KUKA KRL program: dockof_1.src, dockof_1.dat

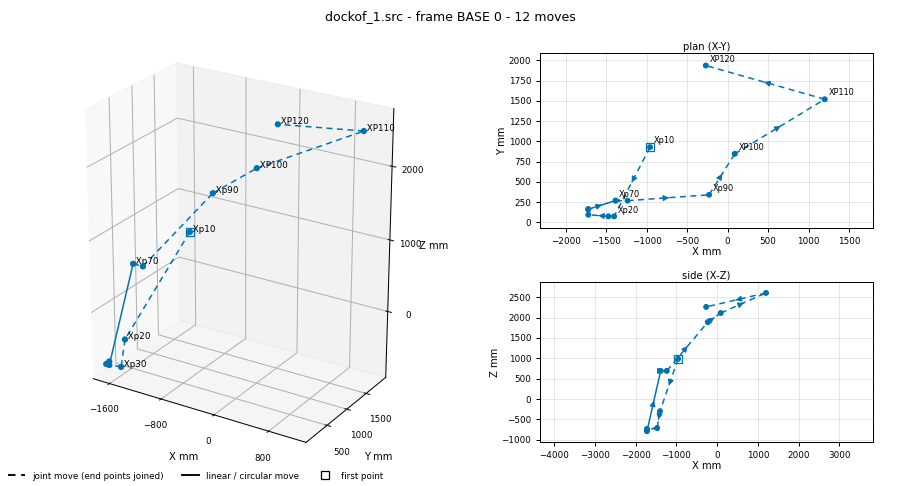
[picture p0: tool path of dockof_1.src in frame BASE 0, 12 of 12 moves have a stored position in this frame; points joined in program order, loops and branches not executed]
--- dockof_1.src ---
&ACCESS RVP1
&REL 140
&COMMENT PLACE GUN 1
DEF DOCKOF_1( )
;================================================
; MODEL    :
; IE GROUP :
; STATION  :
; ROBOT    :
; FUNCTION : DOCK OFF GUN 1
;================================================
;FOLD INI
;FOLD BASISTECH INI
GLOBAL INTERRUPT DECL 3 WHEN $STOPMESS==TRUE DO IR_STOPM ( )
INTERRUPT ON 3
BAS (#INITMOV,0 )
;ENDFOLD (BASISTECH INI)
;FOLD GRIPPERTECH INI
USER_GRP(0,DUMMY,DUMMY,GDEFAULT)
;ENDFOLD (GRIPPERTECH INI)
;FOLD USER INI
;Make your modifications here

;ENDFOLD (USER INI)
;ENDFOLD (INI)

PGNO1_TYPE=0

;FOLD PTP p10 H RETR CLS Gun= 1 Pair= FIRST Tool[1]:Gun 1 Base[0];%{PE}%R 6.0.16,%MKUKATPSPOT,%CRETR,%VPTP,%P 1:PTP, 2:p10, 3:, 5:100, 7:H, 9:#CLO, 11:1, 13:#FIRST
$BWDSTART=FALSE
PDAT_ACT=PH
FDAT_ACT=Fp10
BAS(#PTP_PARAMS,PH.VEL)
S_ACT.GUN=1
S_ACT.PAIR=#FIRST
S_ACT.RETR=#CLO
S_READY=FALSE
TRIGGER WHEN DISTANCE=1 DELAY=0.0 DO USERSPOT(#RETR, S_ACT) PRIO=-1
PTP Xp10
WAIT FOR S_READY
;ENDFOLD

;Open flap 1
;FOLD DOCKING.FLAP_OPN 1 ;%{PE}%MKUKATPUSER
DOCKING (#FLAP_OPN ,1)
;ENDFOLD

;FOLD ; Check docking station 1 ready to dock off;%{PE}%R 2.4.14,%MKUKATPBASIS,%CCOMMENT,%VNORMAL,%P 2:Check docking station 1 ready to dock off
;ENDFOLD
DOCKING (#REQ_DOCK_OFF,1)

;FOLD PTP p20 CONT Vel= 100 % H Tool[1]:Gun 1 Base[0];%{PE}%R 5.4.35,%MKUKATPBASIS,%CMOVE,%VPTP,%P 1:PTP, 2:p20, 3:C_PTP, 5:100, 7:H
$BWDSTART=FALSE
PDAT_ACT=PH
FDAT_ACT=Fp20
BAS(#PTP_PARAMS,100)
PTP Xp20 C_PTP
;ENDFOLD
;FOLD PTP p30 CONT Vel= 100 % H Tool[1]:Gun 1 Base[0];%{PE}%R 5.4.35,%MKUKATPBASIS,%CMOVE,%VPTP,%P 1:PTP, 2:p30, 3:C_PTP, 5:100, 7:H
$BWDSTART=FALSE
PDAT_ACT=PH
FDAT_ACT=Fp30
BAS(#PTP_PARAMS,100)
PTP Xp30 C_PTP
;ENDFOLD

;FOLD ; Above dock position station 1;%{PE}%R 2.4.14,%MKUKATPBASIS,%CCOMMENT,%VNORMAL,%P 2:Above dock position station 1
;ENDFOLD
;FOLD PTP p40  Vel= 100 % H Tool[1]:Gun 1 Base[0];%{PE}%R 5.4.35,%MKUKATPBASIS,%CMOVE,%VPTP,%P 1:PTP, 2:p40, 3:, 5:100, 7:H
$BWDSTART=FALSE
PDAT_ACT=PH
FDAT_ACT=Fp40
BAS(#PTP_PARAMS,100)
PTP Xp40
;ENDFOLD
;FOLD LIN p50  Vel= 0.2 m/s H Tool[1]:Gun 1 Base[0];%{PE}%R 5.4.35,%MKUKATPBASIS,%CMOVE,%VLIN,%P 1:LIN, 2:p50, 3:, 5:0.2, 7:H
$BWDSTART=FALSE
LDAT_ACT=LH
FDAT_ACT=Fp50
BAS(#CP_PARAMS,0.2)
LIN Xp50
;ENDFOLD

;FOLD ; In Dock position Station 1;%{PE}%R 2.4.14,%MKUKATPBASIS,%CCOMMENT,%VNORMAL,%P 2:In Dock position Station 1
;ENDFOLD
;FOLD LIN p60  Vel= 0.2 m/s H Tool[1]:Gun 1 Base[0];%{PE}%R 5.4.35,%MKUKATPBASIS,%CMOVE,%VLIN,%P 1:LIN, 2:p60, 3:, 5:0.2, 7:H
$BWDSTART=FALSE
LDAT_ACT=LH
FDAT_ACT=Fp60
BAS(#CP_PARAMS,0.2)
LIN Xp60
;ENDFOLD

;FOLD ; Unlock Docking plate;%{PE}%R 2.4.14,%MKUKATPBASIS,%CCOMMENT,%VNORMAL,%P 2:Unlock Docking plate
;ENDFOLD
DOCKING (#TOOL_UNLOCK,1)

;FOLD ; Out Docking station 1;%{PE}%R 2.4.14,%MKUKATPBASIS,%CCOMMENT,%VNORMAL,%P 2:Out Docking station 1
;ENDFOLD
;FOLD LIN p70  Vel= 0.2 m/s H Tool[10]:Dock plate Base[0];%{PE}%R 5.4.35,%MKUKATPBASIS,%CMOVE,%VLIN,%P 1:LIN, 2:p70, 3:, 5:0.2, 7:H
$BWDSTART=FALSE
LDAT_ACT=LH
FDAT_ACT=Fp70
BAS(#CP_PARAMS,0.2)
LIN Xp70
;ENDFOLD

;FOLD ; Check docking plate open and station 1 ok;%{PE}%R 2.4.14,%MKUKATPBASIS,%CCOMMENT,%VNORMAL,%P 2:Check docking plate open and station 1 ok
;ENDFOLD
DOCKING (#CHK_TOOL_OFF,1)

;FOLD PTP p80 CONT Vel= 100 % H Tool[10]:Dock plate Base[0];%{PE}%R 5.4.35,%MKUKATPBASIS,%CMOVE,%VPTP,%P 1:PTP, 2:p80, 3:C_PTP, 5:100, 7:H
$BWDSTART=FALSE
PDAT_ACT=PH
FDAT_ACT=Fp80
BAS(#PTP_PARAMS,100)
PTP Xp80 C_PTP
;ENDFOLD
;FOLD PTP p90 CONT Vel= 100 % H Tool[10]:Dock plate Base[0];%{PE}%R 5.4.35,%MKUKATPBASIS,%CMOVE,%VPTP,%P 1:PTP, 2:p90, 3:C_PTP, 5:100, 7:H
$BWDSTART=FALSE
PDAT_ACT=PH
FDAT_ACT=Fp90
BAS(#PTP_PARAMS,100)
PTP Xp90 C_PTP
;ENDFOLD
;FOLD PTP P100 CONT Vel= 100 % H Tool[10]:Dock plate Base[0];%{PE}%R 5.4.35,%MKUKATPBASIS,%CMOVE,%VPTP,%P 1:PTP, 2:P100, 3:C_PTP, 5:100, 7:H
$BWDSTART=FALSE
PDAT_ACT=PH
FDAT_ACT=FP100
BAS(#PTP_PARAMS,100)
PTP XP100 C_PTP
;ENDFOLD
;FOLD PTP P110 CONT Vel= 100 % H Tool[10]:Dock plate Base[0];%{PE}%R 5.4.35,%MKUKATPBASIS,%CMOVE,%VPTP,%P 1:PTP, 2:P110, 3:C_PTP, 5:100, 7:H
$BWDSTART=FALSE
PDAT_ACT=PH
FDAT_ACT=FP110
BAS(#PTP_PARAMS,100)
PTP XP110 C_PTP
;ENDFOLD
;FOLD PTP P120  Vel= 100 % H Tool[10]:Dock plate Base[0];%{PE}%R 5.4.35,%MKUKATPBASIS,%CMOVE,%VPTP,%P 1:PTP, 2:P120, 3:, 5:100, 7:H
$BWDSTART=FALSE
PDAT_ACT=PH
FDAT_ACT=FP120
BAS(#PTP_PARAMS,100)
PTP XP120
;ENDFOLD

;Close flap 1
;FOLD DOCKING.FLAP_CLS 1 ;%{PE}%MKUKATPUSER
DOCKING (#FLAP_CLS ,1)
;ENDFOLD
END

--- dockof_1.dat ---
&ACCESS RVP1
&REL 140
&COMMENT PLACE GUN 1
DEFDAT  DOCKOF_1
;FOLD EXTERNAL DECLARATIONS;%{PE}%MKUKATPBASIS,%CEXT,%VCOMMON,%P
;FOLD GRIPPERTECH EXT
EXT  H50 (INT  :IN,INT  :IN,INT  :IN,GRP_TYP  :IN )
;ENDFOLD (GRIPPERTECH EXT)
;FOLD SPOTTECH EXT
EXT  USERSPOT (S_COMMAND  :IN,SPOT_TYPE  :IN )
;ENDFOLD (SPOTTECH EXT)
;FOLD BASISTECH EXT;%{PE}%MKUKATPBASIS,%CEXT,%VEXT,%P
EXT  BAS (BAS_COMMAND  :IN,REAL  :IN )
DECL INT SUCCESS
;ENDFOLD (BASISTECH EXT)
;FOLD USER EXT;%{E}%MKUKATPUSER,%CEXT,%VEXT,%P
;Make here your modifications
;ENDFOLD (USER EXT)
;ENDFOLD (EXTERNAL DECLERATIONS)
;*      FDAT Declarations     *

;******************************
;*     E6POS Declarations     *
;******************************

DECL E6POS XP10={X -958.092896,Y 929.286072,Z 985.583801,A 92.0790787,B 72.5537262,C -179.835205,S 6,T 26,E1 -2887.177,E2 0.0,E3 0.0,E4 0.0,E5 0.0,E6 0.0}
DECL E6POS XP20={X -1401.91199,Y 74.2533875,Z -298.352112,A 148.144104,B 66.4622421,C -119.998596,S 6,T 26,E1 -2887.177,E2 0.0,E3 0.0,E4 0.0,E5 0.0,E6 0.0}
DECL E6POS XP30={X -1472.677,Y 74.3642273,Z -711.034302,A 124.0728,B 75.2480164,C -145.361298,S 6,T 24,E1 -2887.1709,E2 0.0,E3 0.0,E4 0.0,E5 0.0,E6 0.0}
DECL E6POS XP40={X -1720.43298,Y 93.9440384,Z -744.223206,A 93.5065613,B 77.8009262,C -176.743103,S 6,T 24,E1 -2887.16895,E2 0.0,E3 0.0,E4 0.0,E5 0.0,E6 0.0}
DECL E6POS XP50={X -1721.24402,Y 162.016998,Z -737.295593,A 93.6967621,B 78.4185486,C -176.548294,S 6,T 26,E1 -2887.16602,E2 0.0,E3 0.0,E4 0.0,E5 0.0,E6 0.0}
DECL E6POS XP60={X -1721.22095,Y 162.031906,Z -788.690186,A 93.6951904,B 78.4176025,C -176.550095,S 6,T 24,E1 -2887.16602,E2 0.0,E3 0.0,E4 0.0,E5 0.0,E6 0.0}
DECL E6POS XP70={X -1385.61304,Y 268.545685,Z 690.665405,A -89.8919601,B 60.7910385,C 90.3870926,S 6,T 26,E1 -2887.16211,E2 0.0,E3 0.0,E4 0.0,E5 0.0,E6 0.0}
DECL E6POS XP80={X -1235.49597,Y 267.90979,Z 691.138184,A -89.8916702,B 60.792141,C 90.3865814,S 6,T 26,E1 -2887.16211,E2 0.0,E3 0.0,E4 0.0,E5 0.0,E6 0.0}
DECL E6POS XP90={X -228.028305,Y 340.791901,Z 1887.44702,A -60.9967194,B 52.6837311,C 89.3817062,S 6,T 26,E1 -2702.90991,E2 0.0,E3 0.0,E4 0.0,E5 0.0,E6 0.0}

;******************************
;*     FDAT Declarations      *
;******************************

DECL FDAT FP10={TOOL_NO 1,BASE_NO 0,IPO_FRAME #BASE}
DECL FDAT FP20={TOOL_NO 1,BASE_NO 0,IPO_FRAME #BASE}
DECL FDAT FP30={TOOL_NO 1,BASE_NO 0,IPO_FRAME #BASE}
DECL FDAT FP40={TOOL_NO 1,BASE_NO 0,IPO_FRAME #BASE}
DECL FDAT FP50={TOOL_NO 1,BASE_NO 0,IPO_FRAME #BASE}
DECL FDAT FP60={TOOL_NO 1,BASE_NO 0,IPO_FRAME #BASE}
DECL FDAT FP70={TOOL_NO 10,BASE_NO 0,IPO_FRAME #BASE}
DECL FDAT FP80={TOOL_NO 10,BASE_NO 0,IPO_FRAME #BASE}
DECL FDAT FP90={TOOL_NO 10,BASE_NO 0,IPO_FRAME #BASE}

;******************************
;*  PDAT & LDAT Declarations  *
;******************************

DECL PDAT PH={VEL 100.0,ACC 100.0,APO_DIST 100.0}
DECL LDAT LH={VEL 2.0,ACC 100.0,APO_DIST 100.0,APO_FAC 50.0,ORI_TYP #VAR}

DECL E6POS XP100={X 89.4917221,Y 846.667114,Z 2110.875,A -45.7969208,B 48.727829,C 88.0354996,S 6,T 26,E1 -2602.28296,E2 0.0,E3 0.0,E4 0.0,E5 0.0,E6 0.0}
DECL FDAT FP100={TOOL_NO 10,BASE_NO 0,IPO_FRAME #BASE,POINT2[] " "}
DECL E6POS XP110={X 1200.62598,Y 1521.23999,Z 2604.01294,A 24.9274902,B 16.2740307,C 74.0746231,S 6,T 27,E1 -1873.25098,E2 0.0,E3 0.0,E4 0.0,E5 0.0,E6 0.0}
DECL FDAT FP110={TOOL_NO 10,BASE_NO 0,IPO_FRAME #BASE,POINT2[] " "}
DECL E6POS XP120={X -268.902893,Y 1937.71204,Z 2261.58301,A 150.224106,B 20.9240704,C 81.1927032,S 6,T 59,E1 -735.491699,E2 0.0,E3 0.0,E4 0.0,E5 0.0,E6 0.0}
DECL FDAT FP120={TOOL_NO 10,BASE_NO 0,IPO_FRAME #BASE,POINT2[] " "}
DECL E6POS XP130={X -679.041687,Y 1849.04199,Z 1006.25299,A -155.049393,B -0.176348105,C -178.604294,S 2,T 43,E1 -735.489929,E2 0.0,E3 0.0,E4 0.0,E5 0.0,E6 0.0}
DECL FDAT FP130={TOOL_NO 10,BASE_NO 0,IPO_FRAME #BASE,POINT2[] " "}
DECL E6POS XP15={X -1085.271,Y -265.315704,Z -103.108398,A 95.7909622,B 76.2946014,C -174.720093,S 6,T 26,E1 -2665.03003,E2 0.0,E3 0.0,E4 0.0,E5 0.0,E6 0.0}
DECL FDAT Fp15={TOOL_NO 1,BASE_NO 0,IPO_FRAME #BASE,POINT2[] " "}
DECL E6POS XP16={X -1720.396,Y -246.031799,Z -744.200378,A 93.5082932,B 77.8141632,C -176.740494,S 6,T 24,E1 -2575.16602,E2 0.0,E3 0.0,E4 0.0,E5 0.0,E6 0.0}
DECL FDAT Fp16={TOOL_NO 1,BASE_NO 0,IPO_FRAME #BASE,POINT2[] " "}
DECL SPOT_SUGG_T LAST_SPOT={GUN[] "1                       ",RETR_CMD[] "#OPN                    ",CHOISE[] "#FIRST                  ",CLO_TM[] "0                       ",PGNO1[] "1                       ",PRESS1[] "0                       ",PGNO2[] "1                       ",PRESS2[] "0                       ",SPOT_PARAMS[] "SDAT0                   "}
DECL BASIS_SUGG_T LAST_BASIS={POINT1[] "p10                     ",POINT2[] "p10                     ",CP_PARAMS[] "CPDAT0                  ",PTP_PARAMS[] "H                       ",CONT[] "                        ",CP_VEL[] "2.0                     ",PTP_VEL[] "100                     "}
ENDDAT
